// Mitsubishi GX Works2 project: MiniFactoryFinal1   PLC: FX2N/FX2NC

PROGRAM MAIN
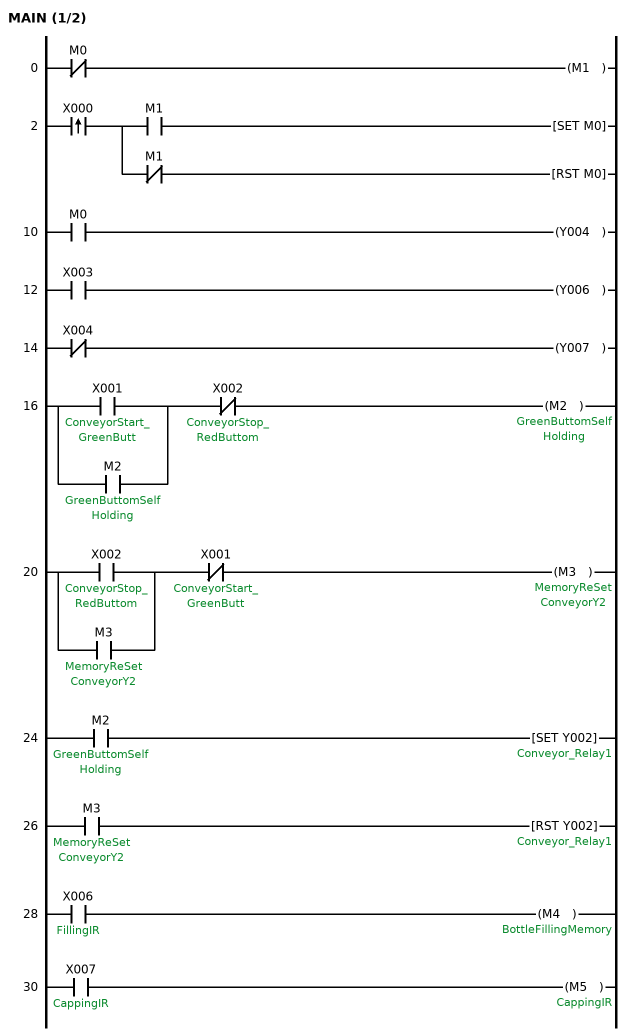
0     LDI     M0
      OUT     M1
2     LDP     X000
      MPS
      AND     M1
      SET     M0
      MPP
      ANI     M1
      RST     M0
10    LD      M0
      OUT     Y004
12    LD      X003
      OUT     Y006
14    LDI     X004
      OUT     Y007
16    LD      X001  ; ConveyorStart_GreenButt
      OR      M2  ; GreenButtomSelfHolding
      ANI     X002  ; ConveyorStop_RedButtom
      OUT     M2  ; GreenButtomSelfHolding
20    LD      X002  ; ConveyorStop_RedButtom
      OR      M3  ; MemoryReSetConveyorY2
      ANI     X001  ; ConveyorStart_GreenButt
      OUT     M3  ; MemoryReSetConveyorY2
24    LD      M2  ; GreenButtomSelfHolding
      SET     Y002  ; Conveyor_Relay1
26    LD      M3  ; MemoryReSetConveyorY2
      RST     Y002  ; Conveyor_Relay1
28    LD      X006  ; FillingIR
      OUT     M4  ; BottleFillingMemory
30    LD      X007  ; CappingIR
      OUT     M5  ; CappingIR
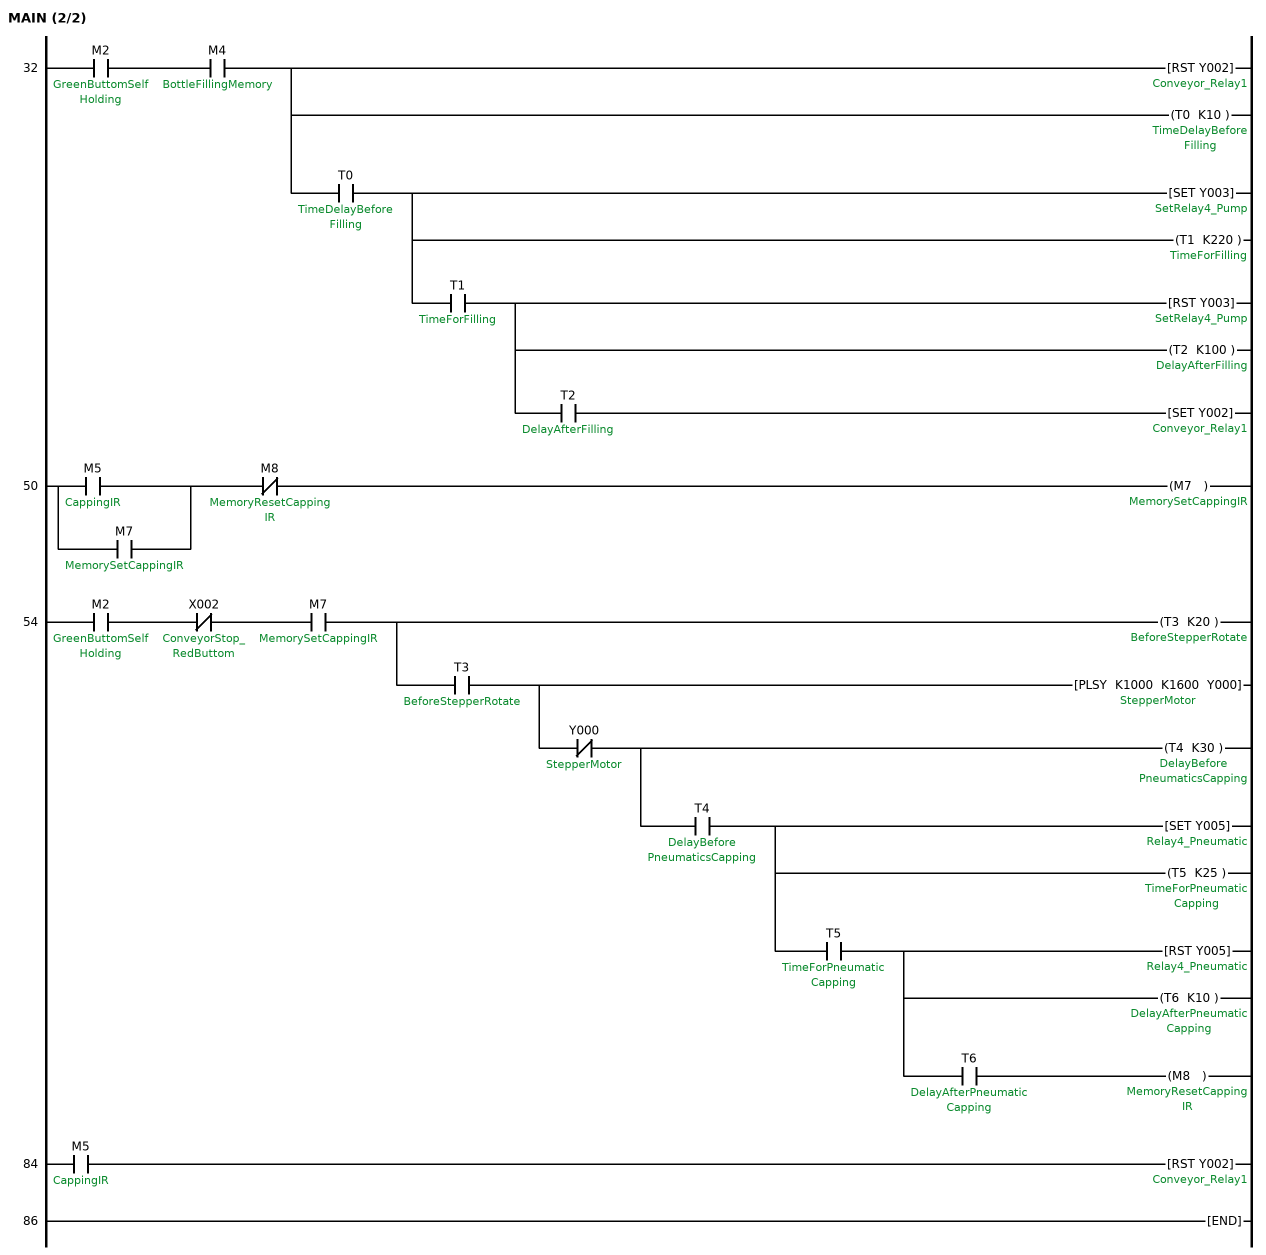
32    LD      M2  ; GreenButtomSelfHolding
      AND     M4  ; BottleFillingMemory
      RST     Y002  ; Conveyor_Relay1
      OUT     T0 K10  ; TimeDelayBeforeFilling
      AND     T0  ; TimeDelayBeforeFilling
      SET     Y003  ; SetRelay4_Pump
      OUT     T1 K220  ; TimeForFilling
      AND     T1  ; TimeForFilling
      RST     Y003  ; SetRelay4_Pump
      OUT     T2 K100  ; DelayAfterFilling
      AND     T2  ; DelayAfterFilling
      SET     Y002  ; Conveyor_Relay1
50    LD      M5  ; CappingIR
      OR      M7  ; MemorySetCappingIR
      ANI     M8  ; MemoryResetCappingIR
      OUT     M7  ; MemorySetCappingIR
54    LD      M2  ; GreenButtomSelfHolding
      ANI     X002  ; ConveyorStop_RedButtom
      AND     M7  ; MemorySetCappingIR
      OUT     T3 K20  ; BeforeStepperRotate
      AND     T3  ; BeforeStepperRotate
      PLSY    K1000 K1600 Y000  ; StepperMotor
      ANI     Y000  ; StepperMotor
      OUT     T4 K30  ; DelayBeforePneumaticsCapping
      AND     T4  ; DelayBeforePneumaticsCapping
      SET     Y005  ; Relay4_Pneumatic
      OUT     T5 K25  ; TimeForPneumaticCapping
      AND     T5  ; TimeForPneumaticCapping
      RST     Y005  ; Relay4_Pneumatic
      OUT     T6 K10  ; DelayAfterPneumaticCapping
      AND     T6  ; DelayAfterPneumaticCapping
      OUT     M8  ; MemoryResetCappingIR
84    LD      M5  ; CappingIR
      RST     Y002  ; Conveyor_Relay1
86    END
END_PROGRAM

// device comments not shown above
M6  ; MemoryResetConveyor
